INTERFACE I_MutBool EXTENDS I_Bool

PROPERTY Val : BOOL
SET
END_SET
END_PROPERTY

END_INTERFACE

(* stored: Version 1.1.0.1
   Itf I_MutBool: Id {4993206b-a094-4215-8882-2d2a8472f22b}
   Property Val: Id {a69d0115-41b6-4a27-966d-624592868abc}
   Set Set: Id {de0c7f51-e567-43e3-bff0-8003b8416474} *)
